REGION Network 23: AXIS W21 MOVE AXIS AND FEED HOLD CONDITIONS
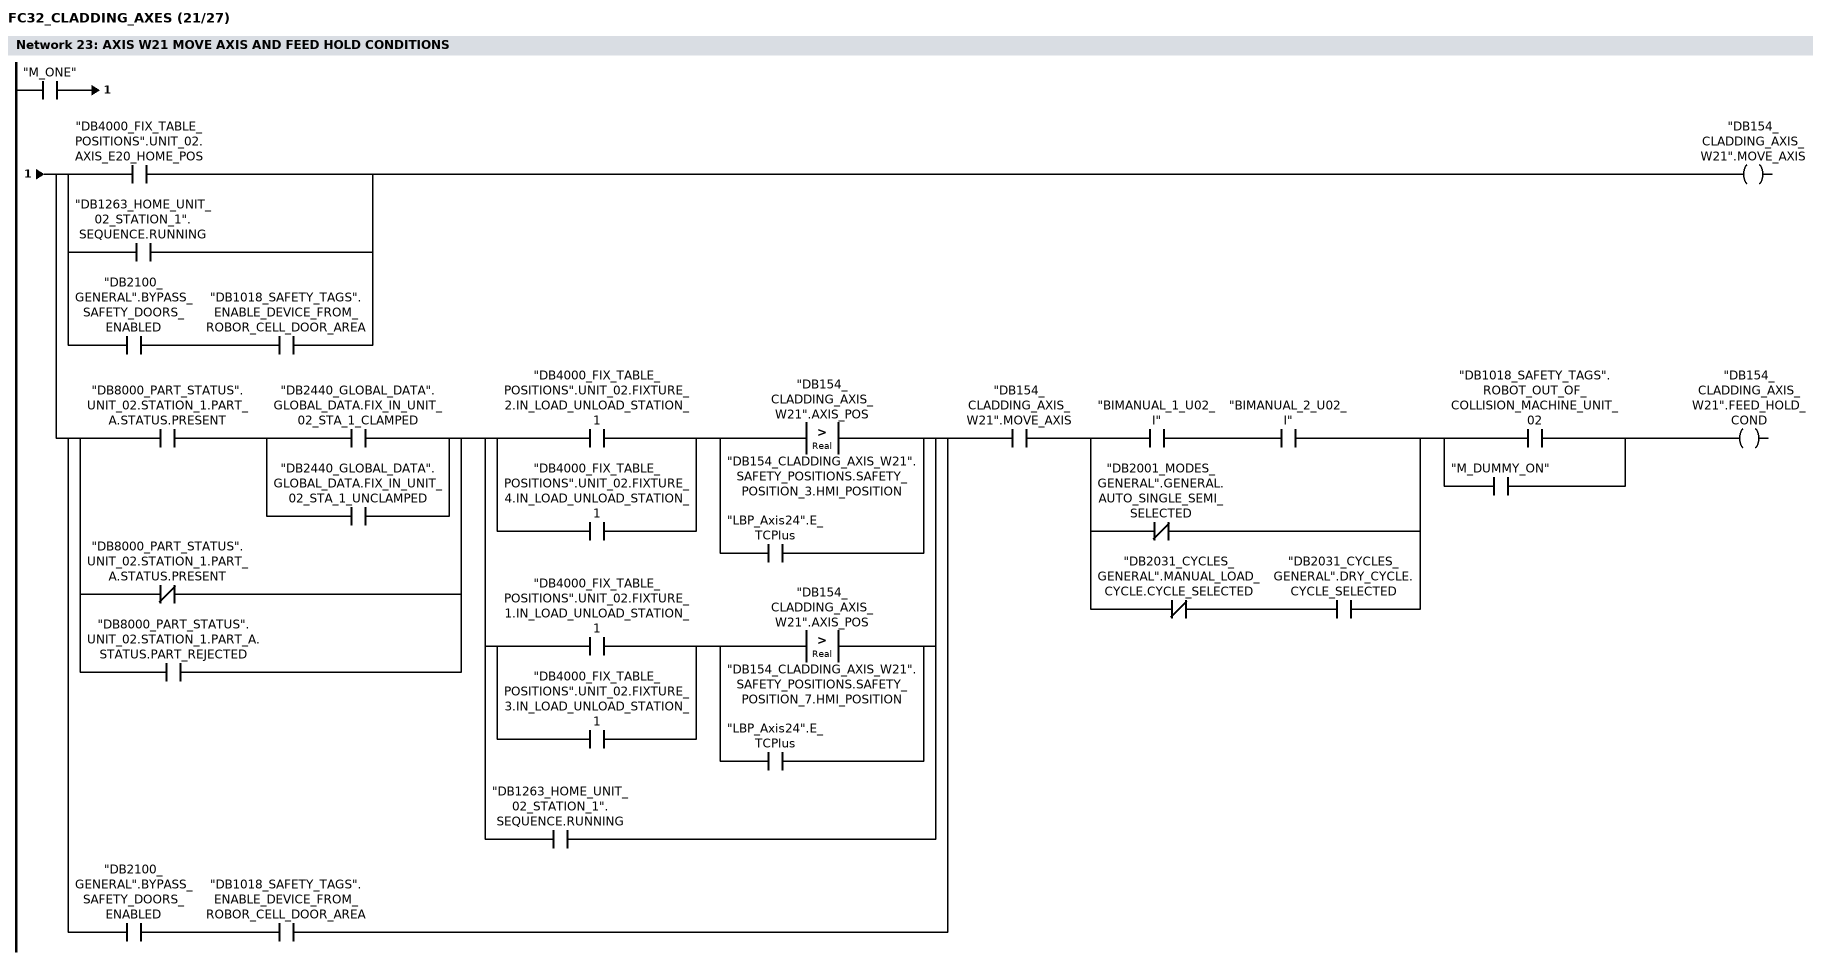
   RUNG wire#powerrail
      Contact( "M_ONE" )
      wire#w1
      Contact( "DB4000_FIX_TABLE_POSITIONS".UNIT_02.AXIS_E20_HOME_POS )
      wire#w2
      Coil( "DB154_CLADDING_AXIS_W21".MOVE_AXIS )
   END_RUNG
   RUNG wire#w1
      Contact( "DB1263_HOME_UNIT_02_STATION_1".SEQUENCE.RUNNING )
   END_RUNG wire#w2
   RUNG wire#w1
      Contact( "DB2100_GENERAL".BYPASS_SAFETY_DOORS_ENABLED )
      Contact( "DB1018_SAFETY_TAGS".ENABLE_DEVICE_FROM_ROBOR_CELL_DOOR_AREA )
   END_RUNG wire#w2
   RUNG wire#w1
      Contact( "DB8000_PART_STATUS".UNIT_02.STATION_1.PART_A.STATUS.PRESENT )
      wire#w3
      Contact( "DB2440_GLOBAL_DATA".GLOBAL_DATA.FIX_IN_UNIT_02_STA_1_CLAMPED )
      wire#w4
      Contact( "DB4000_FIX_TABLE_POSITIONS".UNIT_02.FIXTURE_2.IN_LOAD_UNLOAD_STATION_1 )
      wire#w5
      { S7_Templates := "SrcType := Real" } GT_Contact(in1 := "DB154_CLADDING_AXIS_W21".AXIS_POS, in2 := "DB154_CLADDING_AXIS_W21".SAFETY_POSITIONS.SAFETY_POSITION_3.HMI_POSITION)
      wire#w6
      Contact( "DB154_CLADDING_AXIS_W21".MOVE_AXIS )
      wire#w8
      Contact( "BIMANUAL_1_U02_I" )
      Contact( "BIMANUAL_2_U02_I" )
      wire#w9
      Contact( "DB1018_SAFETY_TAGS".ROBOT_OUT_OF_COLLISION_MACHINE_UNIT_02 )
      wire#w10
      Coil( "DB154_CLADDING_AXIS_W21".FEED_HOLD_COND )
   END_RUNG
   RUNG wire#w3
      Contact( "DB2440_GLOBAL_DATA".GLOBAL_DATA.FIX_IN_UNIT_02_STA_1_UNCLAMPED )
   END_RUNG wire#w4
   RUNG wire#w1
      I_Contact( "DB8000_PART_STATUS".UNIT_02.STATION_1.PART_A.STATUS.PRESENT )
   END_RUNG wire#w4
   RUNG wire#w1
      Contact( "DB8000_PART_STATUS".UNIT_02.STATION_1.PART_A.STATUS.PART_REJECTED )
   END_RUNG wire#w4
   RUNG wire#w4
      Contact( "DB4000_FIX_TABLE_POSITIONS".UNIT_02.FIXTURE_4.IN_LOAD_UNLOAD_STATION_1 )
   END_RUNG wire#w5
   RUNG wire#w5
      Contact( "LBP_Axis24".E_TCPlus )
   END_RUNG wire#w6
   RUNG wire#w4
      Contact( "DB4000_FIX_TABLE_POSITIONS".UNIT_02.FIXTURE_1.IN_LOAD_UNLOAD_STATION_1 )
      wire#w7
      { S7_Templates := "SrcType := Real" } GT_Contact(in1 := "DB154_CLADDING_AXIS_W21".AXIS_POS, in2 := "DB154_CLADDING_AXIS_W21".SAFETY_POSITIONS.SAFETY_POSITION_7.HMI_POSITION)
   END_RUNG wire#w6
   RUNG wire#w4
      Contact( "DB4000_FIX_TABLE_POSITIONS".UNIT_02.FIXTURE_3.IN_LOAD_UNLOAD_STATION_1 )
   END_RUNG wire#w7
   RUNG wire#w7
      Contact( "LBP_Axis24".E_TCPlus )
   END_RUNG wire#w6
   RUNG wire#w4
      Contact( "DB1263_HOME_UNIT_02_STATION_1".SEQUENCE.RUNNING )
   END_RUNG wire#w6
   RUNG wire#w1
      Contact( "DB2100_GENERAL".BYPASS_SAFETY_DOORS_ENABLED )
      Contact( "DB1018_SAFETY_TAGS".ENABLE_DEVICE_FROM_ROBOR_CELL_DOOR_AREA )
   END_RUNG wire#w6
   RUNG wire#w8
      I_Contact( "DB2001_MODES_GENERAL".GENERAL.AUTO_SINGLE_SEMI_SELECTED )
   END_RUNG wire#w9
   RUNG wire#w8
      I_Contact( "DB2031_CYCLES_GENERAL".MANUAL_LOAD_CYCLE.CYCLE_SELECTED )
      Contact( "DB2031_CYCLES_GENERAL".DRY_CYCLE.CYCLE_SELECTED )
   END_RUNG wire#w9
   RUNG wire#w9
      Contact( "M_DUMMY_ON" )
   END_RUNG wire#w10
   // the same network as SCL:
   "DB154_CLADDING_AXIS_W21".MOVE_AXIS := "M_ONE" AND ("DB4000_FIX_TABLE_POSITIONS".UNIT_02.AXIS_E20_HOME_POS OR "DB1263_HOME_UNIT_02_STATION_1".SEQUENCE.RUNNING OR ("DB2100_GENERAL".BYPASS_SAFETY_DOORS_ENABLED AND "DB1018_SAFETY_TAGS".ENABLE_DEVICE_FROM_ROBOR_CELL_DOOR_AREA));
   "DB154_CLADDING_AXIS_W21".FEED_HOLD_COND := "M_ONE" AND (((("DB8000_PART_STATUS".UNIT_02.STATION_1.PART_A.STATUS.PRESENT AND ("DB2440_GLOBAL_DATA".GLOBAL_DATA.FIX_IN_UNIT_02_STA_1_CLAMPED OR "DB2440_GLOBAL_DATA".GLOBAL_DATA.FIX_IN_UNIT_02_STA_1_UNCLAMPED)) OR NOT "DB8000_PART_STATUS".UNIT_02.STATION_1.PART_A.STATUS.PRESENT OR "DB8000_PART_STATUS".UNIT_02.STATION_1.PART_A.STATUS.PART_REJECTED) AND ((("DB4000_FIX_TABLE_POSITIONS".UNIT_02.FIXTURE_2.IN_LOAD_UNLOAD_STATION_1 OR "DB4000_FIX_TABLE_POSITIONS".UNIT_02.FIXTURE_4.IN_LOAD_UNLOAD_STATION_1) AND (("DB154_CLADDING_AXIS_W21".AXIS_POS > "DB154_CLADDING_AXIS_W21".SAFETY_POSITIONS.SAFETY_POSITION_3.HMI_POSITION) OR "LBP_Axis24".E_TCPlus)) OR (("DB4000_FIX_TABLE_POSITIONS".UNIT_02.FIXTURE_1.IN_LOAD_UNLOAD_STATION_1 OR "DB4000_FIX_TABLE_POSITIONS".UNIT_02.FIXTURE_3.IN_LOAD_UNLOAD_STATION_1) AND (("DB154_CLADDING_AXIS_W21".AXIS_POS > "DB154_CLADDING_AXIS_W21".SAFETY_POSITIONS.SAFETY_POSITION_7.HMI_POSITION) OR "LBP_Axis24".E_TCPlus)) OR "DB1263_HOME_UNIT_02_STATION_1".SEQUENCE.RUNNING)) OR ("DB2100_GENERAL".BYPASS_SAFETY_DOORS_ENABLED AND "DB1018_SAFETY_TAGS".ENABLE_DEVICE_FROM_ROBOR_CELL_DOOR_AREA)) AND "DB154_CLADDING_AXIS_W21".MOVE_AXIS AND (("BIMANUAL_1_U02_I" AND "BIMANUAL_2_U02_I") OR NOT "DB2001_MODES_GENERAL".GENERAL.AUTO_SINGLE_SEMI_SELECTED OR (NOT "DB2031_CYCLES_GENERAL".MANUAL_LOAD_CYCLE.CYCLE_SELECTED AND "DB2031_CYCLES_GENERAL".DRY_CYCLE.CYCLE_SELECTED)) AND ("DB1018_SAFETY_TAGS".ROBOT_OUT_OF_COLLISION_MACHINE_UNIT_02 OR "M_DUMMY_ON");
END_REGION

REGION Network 24: CALL FB32 AXIS W21
   // 2#0000_0001 OPTIONS 0 BIT 0 MEASURING SYSTEM 2 OPTION
   // 2#0000_0010 OPTIONS 0 BIT 1 ENABLE FC18 OPTION
   // 2#0000_0100 OPTIONS 0 BIT 2 FC18 EXTERNAL POSITION OPTION
   // 2#0000_1000 OPTIONS 0 BIT 3 AXIS B ENABLE FAULTS OPTION
   // 2#0001_0000 OPTIONS 0 BIT 4 SPARE OPTION
   // 2#0010_0000 OPTIONS 0 BIT 5 SPARE OPTION
   // 2#0100_0000 OPTIONS 0 BIT 6 SPARE OPTION
   // 2#1000_0000 OPTIONS 0 BIT 7 SPARE OPTION
   // 
   // 2#0000_0001 OPTIONS 1 BIT 0 AXIS ROLLER OPTION
   // 2#0000_0010 OPTIONS 1 BIT 1 MASTER AXIS OPTION
   // 2#0000_0100 OPTIONS 1 BIT 2 SLAVE AXIS OPTION
   // 2#0000_1000 OPTIONS 1 BIT 3 MASTER-SLAVE AXES INDEPENDENT MOVEMENT WITH HT10 OPTION
   // 2#0001_0000 OPTIONS 1 BIT 4 GANTRY MODE MASTER AXIS OPTION
   // 2#0010_0000 OPTIONS 1 BIT 5 SPARE OPTION
   // 2#0100_0000 OPTIONS 1 BIT 6 SPARE OPTION
   // 2#1000_0000 OPTIONS 1 BIT 7 SPARE OPTION
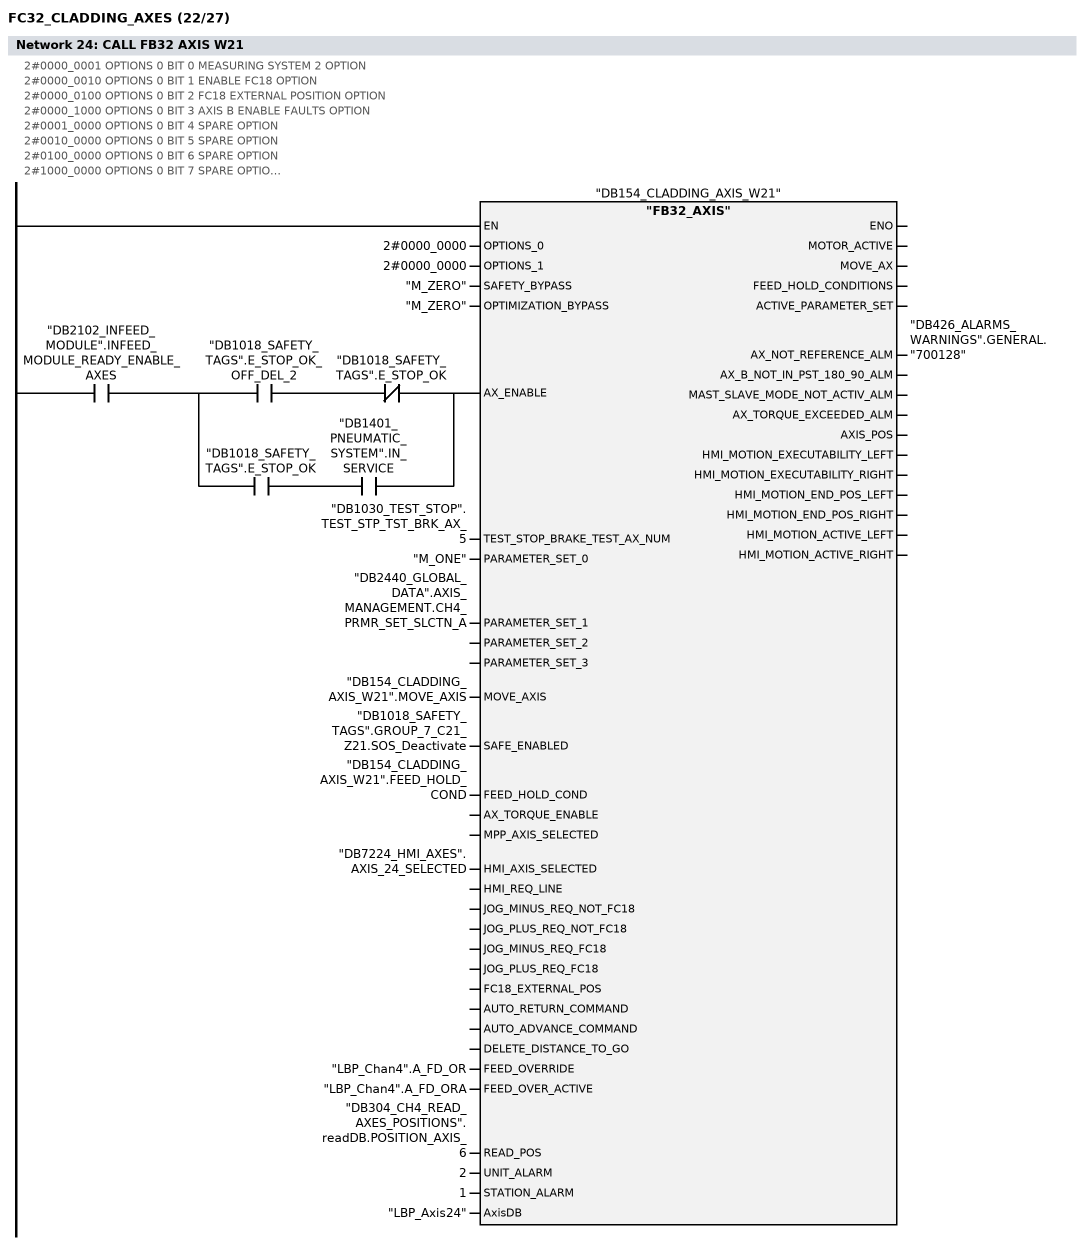
   RUNG wire#powerrail
      "DB154_CLADDING_AXIS_W21"(AX_ENABLE := wire#w2, OPTIONS_0 := 2#0000_0000, OPTIONS_1 := 2#0000_0000, SAFETY_BYPASS := "M_ZERO", OPTIMIZATION_BYPASS := "M_ZERO", TEST_STOP_BRAKE_TEST_AX_NUM := "DB1030_TEST_STOP".TEST_STP_TST_BRK_AX_5, PARAMETER_SET_0 := "M_ONE", PARAMETER_SET_1 := "DB2440_GLOBAL_DATA".AXIS_MANAGEMENT.CH4_PRMR_SET_SLCTN_A, PARAMETER_SET_2 :=, PARAMETER_SET_3 :=, MOVE_AXIS := "DB154_CLADDING_AXIS_W21".MOVE_AXIS, SAFE_ENABLED := "DB1018_SAFETY_TAGS".GROUP_7_C21_Z21.SOS_Deactivate, FEED_HOLD_COND := "DB154_CLADDING_AXIS_W21".FEED_HOLD_COND, AX_TORQUE_ENABLE :=, MPP_AXIS_SELECTED :=, HMI_AXIS_SELECTED := "DB7224_HMI_AXES".AXIS_24_SELECTED, HMI_REQ_LINE :=, JOG_MINUS_REQ_NOT_FC18 :=, JOG_PLUS_REQ_NOT_FC18 :=, JOG_MINUS_REQ_FC18 :=, JOG_PLUS_REQ_FC18 :=, FC18_EXTERNAL_POS :=, AUTO_RETURN_COMMAND :=, AUTO_ADVANCE_COMMAND :=, DELETE_DISTANCE_TO_GO :=, FEED_OVERRIDE := "LBP_Chan4".A_FD_OR, FEED_OVER_ACTIVE := "LBP_Chan4".A_FD_ORA, READ_POS := "DB304_CH4_READ_AXES_POSITIONS".readDB.POSITION_AXIS_6, UNIT_ALARM := 2, STATION_ALARM := 1, AxisDB := "LBP_Axis24", MOTOR_ACTIVE =>, MOVE_AX =>, FEED_HOLD_CONDITIONS =>, ACTIVE_PARAMETER_SET =>, AX_NOT_REFERENCE_ALM => "DB426_ALARMS_WARNINGS".GENERAL."700128", AX_B_NOT_IN_PST_180_90_ALM =>, MAST_SLAVE_MODE_NOT_ACTIV_ALM =>, AX_TORQUE_EXCEEDED_ALM =>, AXIS_POS =>, HMI_MOTION_EXECUTABILITY_LEFT =>, HMI_MOTION_EXECUTABILITY_RIGHT =>, HMI_MOTION_END_POS_LEFT =>, HMI_MOTION_END_POS_RIGHT =>, HMI_MOTION_ACTIVE_LEFT =>, HMI_MOTION_ACTIVE_RIGHT =>)
   END_RUNG
   RUNG wire#powerrail
      Contact( "DB2102_INFEED_MODULE".INFEED_MODULE_READY_ENABLE_AXES )
      wire#w1
      Contact( "DB1018_SAFETY_TAGS".E_STOP_OK_OFF_DEL_2 )
      I_Contact( "DB1018_SAFETY_TAGS".E_STOP_OK )
   END_RUNG wire#w2
   RUNG wire#w1
      Contact( "DB1018_SAFETY_TAGS".E_STOP_OK )
      Contact( "DB1401_PNEUMATIC_SYSTEM".IN_SERVICE )
   END_RUNG wire#w2
   // the same network as SCL:
   "DB154_CLADDING_AXIS_W21"(OPTIONS_0 := 2#0000_0000,   // "FB32_AXIS"
                           OPTIONS_1 := 2#0000_0000,
                           SAFETY_BYPASS := "M_ZERO",
                           OPTIMIZATION_BYPASS := "M_ZERO",
                           AX_ENABLE := "DB2102_INFEED_MODULE".INFEED_MODULE_READY_ENABLE_AXES AND (("DB1018_SAFETY_TAGS".E_STOP_OK_OFF_DEL_2 AND NOT "DB1018_SAFETY_TAGS".E_STOP_OK) OR ("DB1018_SAFETY_TAGS".E_STOP_OK AND "DB1401_PNEUMATIC_SYSTEM".IN_SERVICE)),
                           TEST_STOP_BRAKE_TEST_AX_NUM := "DB1030_TEST_STOP".TEST_STP_TST_BRK_AX_5,
                           PARAMETER_SET_0 := "M_ONE",
                           PARAMETER_SET_1 := "DB2440_GLOBAL_DATA".AXIS_MANAGEMENT.CH4_PRMR_SET_SLCTN_A,
                           MOVE_AXIS := "DB154_CLADDING_AXIS_W21".MOVE_AXIS,
                           SAFE_ENABLED := "DB1018_SAFETY_TAGS".GROUP_7_C21_Z21.SOS_Deactivate,
                           FEED_HOLD_COND := "DB154_CLADDING_AXIS_W21".FEED_HOLD_COND,
                           HMI_AXIS_SELECTED := "DB7224_HMI_AXES".AXIS_24_SELECTED,
                           FEED_OVERRIDE := "LBP_Chan4".A_FD_OR,
                           FEED_OVER_ACTIVE := "LBP_Chan4".A_FD_ORA,
                           READ_POS := "DB304_CH4_READ_AXES_POSITIONS".readDB.POSITION_AXIS_6,
                           UNIT_ALARM := 2,
                           STATION_ALARM := 1,
                           AxisDB := "LBP_Axis24",
                           AX_NOT_REFERENCE_ALM => "DB426_ALARMS_WARNINGS".GENERAL."700128");
END_REGION

REGION Network 25: AXIS W21 OPERATOR HELP
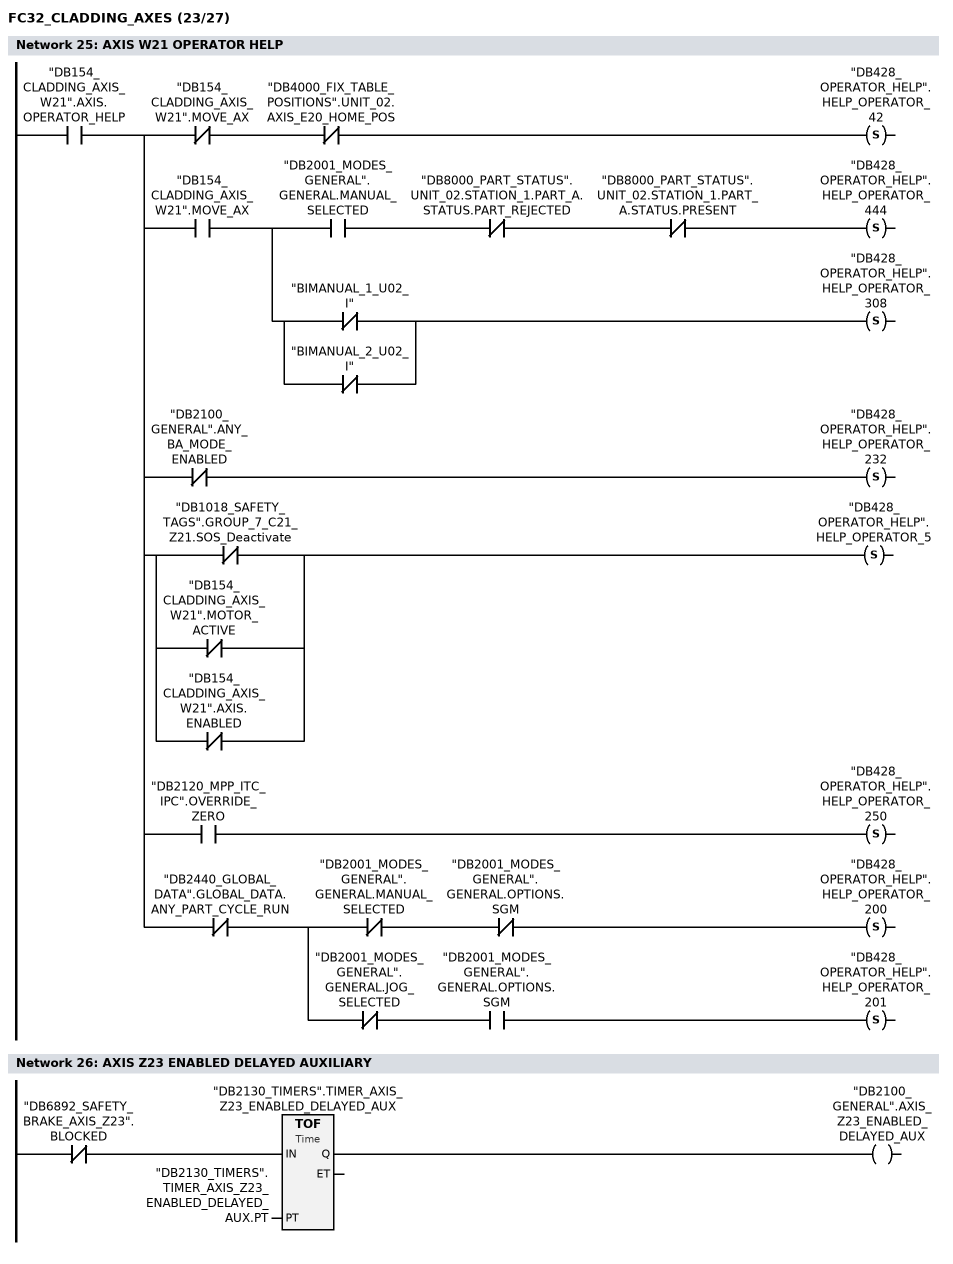
   RUNG wire#powerrail
      Contact( "DB154_CLADDING_AXIS_W21".AXIS.OPERATOR_HELP )
      wire#w1
      I_Contact( "DB154_CLADDING_AXIS_W21".MOVE_AX )
      I_Contact( "DB4000_FIX_TABLE_POSITIONS".UNIT_02.AXIS_E20_HOME_POS )
      S_Coil( "DB428_OPERATOR_HELP".HELP_OPERATOR_42 )
   END_RUNG
   RUNG wire#w1
      Contact( "DB154_CLADDING_AXIS_W21".MOVE_AX )
      wire#w2
      Contact( "DB2001_MODES_GENERAL".GENERAL.MANUAL_SELECTED )
      I_Contact( "DB8000_PART_STATUS".UNIT_02.STATION_1.PART_A.STATUS.PART_REJECTED )
      I_Contact( "DB8000_PART_STATUS".UNIT_02.STATION_1.PART_A.STATUS.PRESENT )
      S_Coil( "DB428_OPERATOR_HELP".HELP_OPERATOR_444 )
   END_RUNG
   RUNG wire#w2
      I_Contact( "BIMANUAL_1_U02_I" )
      wire#w3
      S_Coil( "DB428_OPERATOR_HELP".HELP_OPERATOR_308 )
   END_RUNG
   RUNG wire#w2
      I_Contact( "BIMANUAL_2_U02_I" )
   END_RUNG wire#w3
   RUNG wire#w1
      I_Contact( "DB2100_GENERAL".ANY_BA_MODE_ENABLED )
      S_Coil( "DB428_OPERATOR_HELP".HELP_OPERATOR_232 )
   END_RUNG
   RUNG wire#w1
      I_Contact( "DB1018_SAFETY_TAGS".GROUP_7_C21_Z21.SOS_Deactivate )
      wire#w4
      S_Coil( "DB428_OPERATOR_HELP".HELP_OPERATOR_5 )
   END_RUNG
   RUNG wire#w1
      I_Contact( "DB154_CLADDING_AXIS_W21".MOTOR_ACTIVE )
   END_RUNG wire#w4
   RUNG wire#w1
      I_Contact( "DB154_CLADDING_AXIS_W21".AXIS.ENABLED )
   END_RUNG wire#w4
   RUNG wire#w1
      Contact( "DB2120_MPP_ITC_IPC".OVERRIDE_ZERO )
      S_Coil( "DB428_OPERATOR_HELP".HELP_OPERATOR_250 )
   END_RUNG
   RUNG wire#w1
      I_Contact( "DB2440_GLOBAL_DATA".GLOBAL_DATA.ANY_PART_CYCLE_RUN )
      wire#w5
      I_Contact( "DB2001_MODES_GENERAL".GENERAL.MANUAL_SELECTED )
      I_Contact( "DB2001_MODES_GENERAL".GENERAL.OPTIONS.SGM )
      S_Coil( "DB428_OPERATOR_HELP".HELP_OPERATOR_200 )
   END_RUNG
   RUNG wire#w5
      I_Contact( "DB2001_MODES_GENERAL".GENERAL.JOG_SELECTED )
      Contact( "DB2001_MODES_GENERAL".GENERAL.OPTIONS.SGM )
      S_Coil( "DB428_OPERATOR_HELP".HELP_OPERATOR_201 )
   END_RUNG
   // the same network as SCL:
   IF "DB154_CLADDING_AXIS_W21".AXIS.OPERATOR_HELP AND NOT "DB154_CLADDING_AXIS_W21".MOVE_AX AND NOT "DB4000_FIX_TABLE_POSITIONS".UNIT_02.AXIS_E20_HOME_POS THEN
       "DB428_OPERATOR_HELP".HELP_OPERATOR_42 := TRUE;
   END_IF;
   #_w1 := "DB154_CLADDING_AXIS_W21".AXIS.OPERATOR_HELP AND "DB154_CLADDING_AXIS_W21".MOVE_AX;
   IF #_w1 AND "DB2001_MODES_GENERAL".GENERAL.MANUAL_SELECTED AND NOT "DB8000_PART_STATUS".UNIT_02.STATION_1.PART_A.STATUS.PART_REJECTED AND NOT "DB8000_PART_STATUS".UNIT_02.STATION_1.PART_A.STATUS.PRESENT THEN
       "DB428_OPERATOR_HELP".HELP_OPERATOR_444 := TRUE;
   END_IF;
   IF #_w1 AND (NOT "BIMANUAL_1_U02_I" OR NOT "BIMANUAL_2_U02_I") THEN
       "DB428_OPERATOR_HELP".HELP_OPERATOR_308 := TRUE;
   END_IF;
   IF "DB154_CLADDING_AXIS_W21".AXIS.OPERATOR_HELP AND NOT "DB2100_GENERAL".ANY_BA_MODE_ENABLED THEN
       "DB428_OPERATOR_HELP".HELP_OPERATOR_232 := TRUE;
   END_IF;
   IF "DB154_CLADDING_AXIS_W21".AXIS.OPERATOR_HELP AND (NOT "DB1018_SAFETY_TAGS".GROUP_7_C21_Z21.SOS_Deactivate OR NOT "DB154_CLADDING_AXIS_W21".MOTOR_ACTIVE OR NOT "DB154_CLADDING_AXIS_W21".AXIS.ENABLED) THEN
       "DB428_OPERATOR_HELP".HELP_OPERATOR_5 := TRUE;
   END_IF;
   IF "DB154_CLADDING_AXIS_W21".AXIS.OPERATOR_HELP AND "DB2120_MPP_ITC_IPC".OVERRIDE_ZERO THEN
       "DB428_OPERATOR_HELP".HELP_OPERATOR_250 := TRUE;
   END_IF;
   #_w2 := "DB154_CLADDING_AXIS_W21".AXIS.OPERATOR_HELP AND NOT "DB2440_GLOBAL_DATA".GLOBAL_DATA.ANY_PART_CYCLE_RUN;
   IF #_w2 AND NOT "DB2001_MODES_GENERAL".GENERAL.MANUAL_SELECTED AND NOT "DB2001_MODES_GENERAL".GENERAL.OPTIONS.SGM THEN
       "DB428_OPERATOR_HELP".HELP_OPERATOR_200 := TRUE;
   END_IF;
   IF #_w2 AND NOT "DB2001_MODES_GENERAL".GENERAL.JOG_SELECTED AND "DB2001_MODES_GENERAL".GENERAL.OPTIONS.SGM THEN
       "DB428_OPERATOR_HELP".HELP_OPERATOR_201 := TRUE;
   END_IF;
END_REGION

REGION Network 26: AXIS Z23 ENABLED DELAYED AUXILIARY
   RUNG wire#powerrail
      I_Contact( "DB6892_SAFETY_BRAKE_AXIS_Z23".BLOCKED )
      { S7_Templates := "time_type := Time" } "DB2130_TIMERS".TIMER_AXIS_Z23_ENABLED_DELAYED_AUX.TOF(pt := "DB2130_TIMERS".TIMER_AXIS_Z23_ENABLED_DELAYED_AUX.PT, et =>)
      Coil( "DB2100_GENERAL".AXIS_Z23_ENABLED_DELAYED_AUX )
   END_RUNG
   // the same network as SCL:
   "DB2130_TIMERS".TIMER_AXIS_Z23_ENABLED_DELAYED_AUX.TOF(IN := NOT "DB6892_SAFETY_BRAKE_AXIS_Z23".BLOCKED,
                           PT := "DB2130_TIMERS".TIMER_AXIS_Z23_ENABLED_DELAYED_AUX.PT);
   "DB2100_GENERAL".AXIS_Z23_ENABLED_DELAYED_AUX := "DB2130_TIMERS".TIMER_AXIS_Z23_ENABLED_DELAYED_AUX.Q;
END_REGION

REGION Network 27: AXIS Z23 MOVE AXIS AND FEED HOLD CONDITIONS
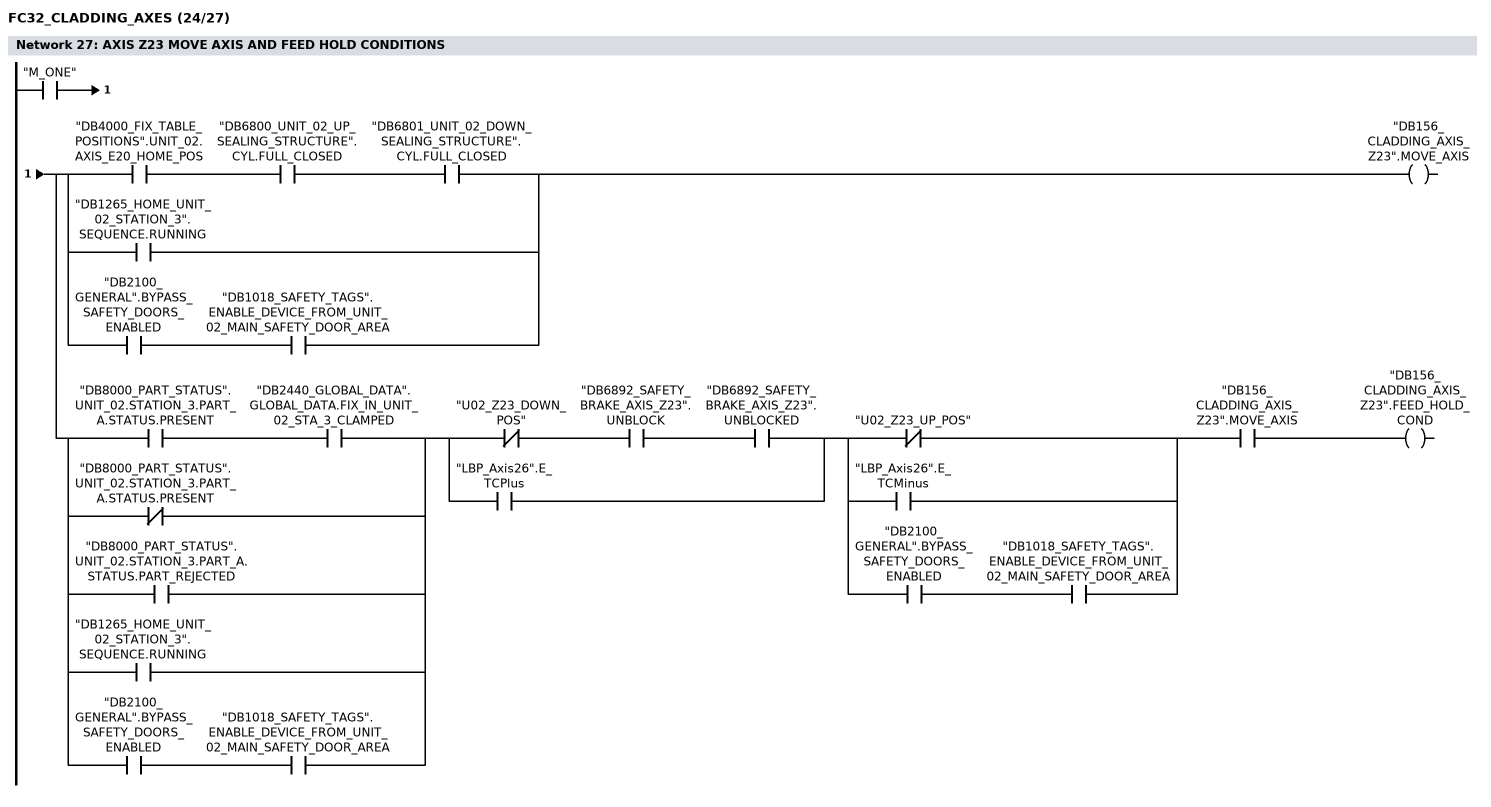
   RUNG wire#powerrail
      Contact( "M_ONE" )
      wire#w1
      Contact( "DB4000_FIX_TABLE_POSITIONS".UNIT_02.AXIS_E20_HOME_POS )
      Contact( "DB6800_UNIT_02_UP_SEALING_STRUCTURE".CYL.FULL_CLOSED )
      Contact( "DB6801_UNIT_02_DOWN_SEALING_STRUCTURE".CYL.FULL_CLOSED )
      wire#w2
      Coil( "DB156_CLADDING_AXIS_Z23".MOVE_AXIS )
   END_RUNG
   RUNG wire#w1
      Contact( "DB1265_HOME_UNIT_02_STATION_3".SEQUENCE.RUNNING )
   END_RUNG wire#w2
   RUNG wire#w1
      Contact( "DB2100_GENERAL".BYPASS_SAFETY_DOORS_ENABLED )
      Contact( "DB1018_SAFETY_TAGS".ENABLE_DEVICE_FROM_UNIT_02_MAIN_SAFETY_DOOR_AREA )
   END_RUNG wire#w2
   RUNG wire#w1
      Contact( "DB8000_PART_STATUS".UNIT_02.STATION_3.PART_A.STATUS.PRESENT )
      Contact( "DB2440_GLOBAL_DATA".GLOBAL_DATA.FIX_IN_UNIT_02_STA_3_CLAMPED )
      wire#w3
      I_Contact( "U02_Z23_DOWN_POS" )
      Contact( "DB6892_SAFETY_BRAKE_AXIS_Z23".UNBLOCK )
      Contact( "DB6892_SAFETY_BRAKE_AXIS_Z23".UNBLOCKED )
      wire#w4
      I_Contact( "U02_Z23_UP_POS" )
      wire#w5
      Contact( "DB156_CLADDING_AXIS_Z23".MOVE_AXIS )
      Coil( "DB156_CLADDING_AXIS_Z23".FEED_HOLD_COND )
   END_RUNG
   RUNG wire#w1
      I_Contact( "DB8000_PART_STATUS".UNIT_02.STATION_3.PART_A.STATUS.PRESENT )
   END_RUNG wire#w3
   RUNG wire#w1
      Contact( "DB8000_PART_STATUS".UNIT_02.STATION_3.PART_A.STATUS.PART_REJECTED )
   END_RUNG wire#w3
   RUNG wire#w1
      Contact( "DB1265_HOME_UNIT_02_STATION_3".SEQUENCE.RUNNING )
   END_RUNG wire#w3
   RUNG wire#w1
      Contact( "DB2100_GENERAL".BYPASS_SAFETY_DOORS_ENABLED )
      Contact( "DB1018_SAFETY_TAGS".ENABLE_DEVICE_FROM_UNIT_02_MAIN_SAFETY_DOOR_AREA )
   END_RUNG wire#w3
   RUNG wire#w3
      Contact( "LBP_Axis26".E_TCPlus )
   END_RUNG wire#w4
   RUNG wire#w4
      Contact( "LBP_Axis26".E_TCMinus )
   END_RUNG wire#w5
   RUNG wire#w4
      Contact( "DB2100_GENERAL".BYPASS_SAFETY_DOORS_ENABLED )
      Contact( "DB1018_SAFETY_TAGS".ENABLE_DEVICE_FROM_UNIT_02_MAIN_SAFETY_DOOR_AREA )
   END_RUNG wire#w5
   // the same network as SCL:
   "DB156_CLADDING_AXIS_Z23".MOVE_AXIS := "M_ONE" AND (("DB4000_FIX_TABLE_POSITIONS".UNIT_02.AXIS_E20_HOME_POS AND "DB6800_UNIT_02_UP_SEALING_STRUCTURE".CYL.FULL_CLOSED AND "DB6801_UNIT_02_DOWN_SEALING_STRUCTURE".CYL.FULL_CLOSED) OR "DB1265_HOME_UNIT_02_STATION_3".SEQUENCE.RUNNING OR ("DB2100_GENERAL".BYPASS_SAFETY_DOORS_ENABLED AND "DB1018_SAFETY_TAGS".ENABLE_DEVICE_FROM_UNIT_02_MAIN_SAFETY_DOOR_AREA));
   "DB156_CLADDING_AXIS_Z23".FEED_HOLD_COND := "M_ONE" AND (("DB8000_PART_STATUS".UNIT_02.STATION_3.PART_A.STATUS.PRESENT AND "DB2440_GLOBAL_DATA".GLOBAL_DATA.FIX_IN_UNIT_02_STA_3_CLAMPED) OR NOT "DB8000_PART_STATUS".UNIT_02.STATION_3.PART_A.STATUS.PRESENT OR "DB8000_PART_STATUS".UNIT_02.STATION_3.PART_A.STATUS.PART_REJECTED OR "DB1265_HOME_UNIT_02_STATION_3".SEQUENCE.RUNNING OR ("DB2100_GENERAL".BYPASS_SAFETY_DOORS_ENABLED AND "DB1018_SAFETY_TAGS".ENABLE_DEVICE_FROM_UNIT_02_MAIN_SAFETY_DOOR_AREA)) AND ((NOT "U02_Z23_DOWN_POS" AND "DB6892_SAFETY_BRAKE_AXIS_Z23".UNBLOCK AND "DB6892_SAFETY_BRAKE_AXIS_Z23".UNBLOCKED) OR "LBP_Axis26".E_TCPlus) AND (NOT "U02_Z23_UP_POS" OR "LBP_Axis26".E_TCMinus OR ("DB2100_GENERAL".BYPASS_SAFETY_DOORS_ENABLED AND "DB1018_SAFETY_TAGS".ENABLE_DEVICE_FROM_UNIT_02_MAIN_SAFETY_DOOR_AREA)) AND "DB156_CLADDING_AXIS_Z23".MOVE_AXIS;
END_REGION

REGION Network 28: CALL FB32 AXIS Z23
   // 2#0000_0001 OPTIONS 0 BIT 0 MEASURING SYSTEM 2 OPTION
   // 2#0000_0010 OPTIONS 0 BIT 1 ENABLE FC18 OPTION
   // 2#0000_0100 OPTIONS 0 BIT 2 FC18 EXTERNAL POSITION OPTION
   // 2#0000_1000 OPTIONS 0 BIT 3 AXIS B ENABLE FAULTS OPTION
   // 2#0001_0000 OPTIONS 0 BIT 4 SPARE OPTION
   // 2#0010_0000 OPTIONS 0 BIT 5 SPARE OPTION
   // 2#0100_0000 OPTIONS 0 BIT 6 SPARE OPTION
   // 2#1000_0000 OPTIONS 0 BIT 7 SPARE OPTION
   // 
   // 2#0000_0001 OPTIONS 1 BIT 0 AXIS ROLLER OPTION
   // 2#0000_0010 OPTIONS 1 BIT 1 MASTER AXIS OPTION
   // 2#0000_0100 OPTIONS 1 BIT 2 SLAVE AXIS OPTION
   // 2#0000_1000 OPTIONS 1 BIT 3 MASTER-SLAVE AXES INDEPENDENT MOVEMENT WITH HT10 OPTION
   // 2#0001_0000 OPTIONS 1 BIT 4 GANTRY MODE MASTER AXIS OPTION
   // 2#0010_0000 OPTIONS 1 BIT 5 SPARE OPTION
   // 2#0100_0000 OPTIONS 1 BIT 6 SPARE OPTION
   // 2#1000_0000 OPTIONS 1 BIT 7 SPARE OPTION
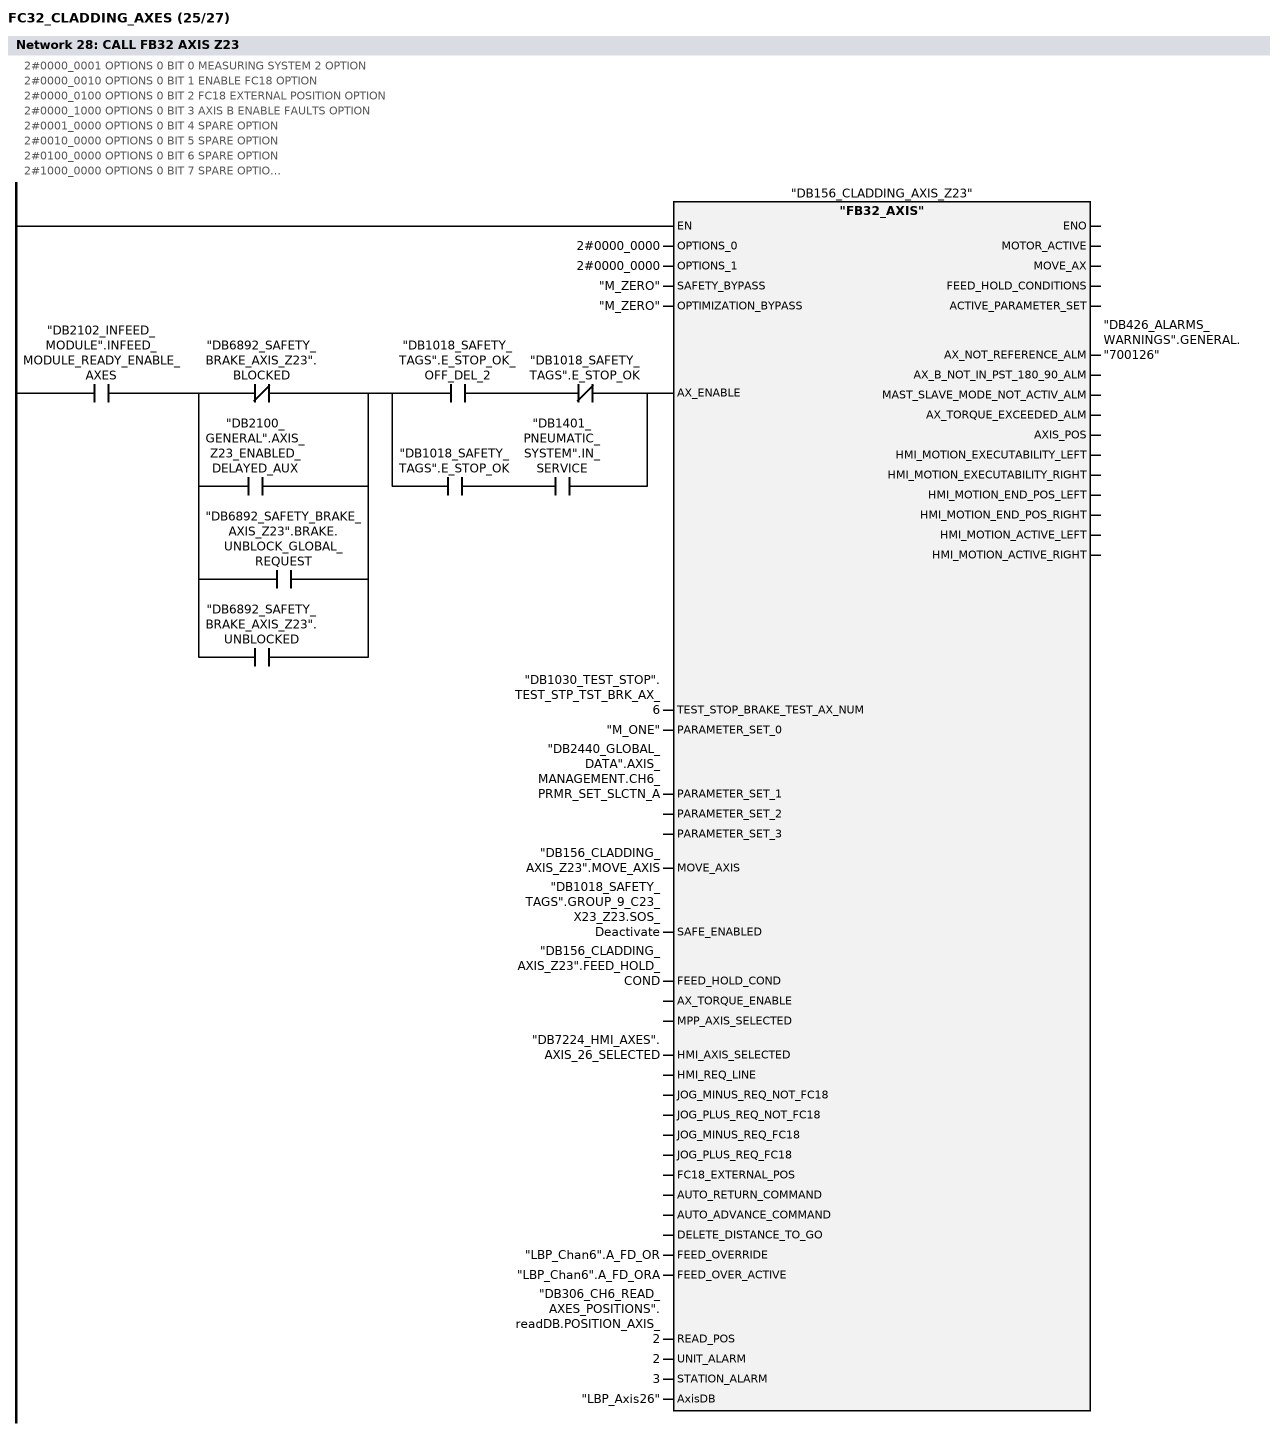
   RUNG wire#powerrail
      "DB156_CLADDING_AXIS_Z23"(AX_ENABLE := wire#w3, OPTIONS_0 := 2#0000_0000, OPTIONS_1 := 2#0000_0000, SAFETY_BYPASS := "M_ZERO", OPTIMIZATION_BYPASS := "M_ZERO", TEST_STOP_BRAKE_TEST_AX_NUM := "DB1030_TEST_STOP".TEST_STP_TST_BRK_AX_6, PARAMETER_SET_0 := "M_ONE", PARAMETER_SET_1 := "DB2440_GLOBAL_DATA".AXIS_MANAGEMENT.CH6_PRMR_SET_SLCTN_A, PARAMETER_SET_2 :=, PARAMETER_SET_3 :=, MOVE_AXIS := "DB156_CLADDING_AXIS_Z23".MOVE_AXIS, SAFE_ENABLED := "DB1018_SAFETY_TAGS".GROUP_9_C23_X23_Z23.SOS_Deactivate, FEED_HOLD_COND := "DB156_CLADDING_AXIS_Z23".FEED_HOLD_COND, AX_TORQUE_ENABLE :=, MPP_AXIS_SELECTED :=, HMI_AXIS_SELECTED := "DB7224_HMI_AXES".AXIS_26_SELECTED, HMI_REQ_LINE :=, JOG_MINUS_REQ_NOT_FC18 :=, JOG_PLUS_REQ_NOT_FC18 :=, JOG_MINUS_REQ_FC18 :=, JOG_PLUS_REQ_FC18 :=, FC18_EXTERNAL_POS :=, AUTO_RETURN_COMMAND :=, AUTO_ADVANCE_COMMAND :=, DELETE_DISTANCE_TO_GO :=, FEED_OVERRIDE := "LBP_Chan6".A_FD_OR, FEED_OVER_ACTIVE := "LBP_Chan6".A_FD_ORA, READ_POS := "DB306_CH6_READ_AXES_POSITIONS".readDB.POSITION_AXIS_2, UNIT_ALARM := 2, STATION_ALARM := 3, AxisDB := "LBP_Axis26", MOTOR_ACTIVE =>, MOVE_AX =>, FEED_HOLD_CONDITIONS =>, ACTIVE_PARAMETER_SET =>, AX_NOT_REFERENCE_ALM => "DB426_ALARMS_WARNINGS".GENERAL."700126", AX_B_NOT_IN_PST_180_90_ALM =>, MAST_SLAVE_MODE_NOT_ACTIV_ALM =>, AX_TORQUE_EXCEEDED_ALM =>, AXIS_POS =>, HMI_MOTION_EXECUTABILITY_LEFT =>, HMI_MOTION_EXECUTABILITY_RIGHT =>, HMI_MOTION_END_POS_LEFT =>, HMI_MOTION_END_POS_RIGHT =>, HMI_MOTION_ACTIVE_LEFT =>, HMI_MOTION_ACTIVE_RIGHT =>)
   END_RUNG
   RUNG wire#powerrail
      Contact( "DB2102_INFEED_MODULE".INFEED_MODULE_READY_ENABLE_AXES )
      wire#w1
      I_Contact( "DB6892_SAFETY_BRAKE_AXIS_Z23".BLOCKED )
      wire#w2
      Contact( "DB1018_SAFETY_TAGS".E_STOP_OK_OFF_DEL_2 )
      I_Contact( "DB1018_SAFETY_TAGS".E_STOP_OK )
   END_RUNG wire#w3
   RUNG wire#w1
      Contact( "DB2100_GENERAL".AXIS_Z23_ENABLED_DELAYED_AUX )
   END_RUNG wire#w2
   RUNG wire#w1
      Contact( "DB6892_SAFETY_BRAKE_AXIS_Z23".BRAKE.UNBLOCK_GLOBAL_REQUEST )
   END_RUNG wire#w2
   RUNG wire#w1
      Contact( "DB6892_SAFETY_BRAKE_AXIS_Z23".UNBLOCKED )
   END_RUNG wire#w2
   RUNG wire#w2
      Contact( "DB1018_SAFETY_TAGS".E_STOP_OK )
      Contact( "DB1401_PNEUMATIC_SYSTEM".IN_SERVICE )
   END_RUNG wire#w3
   // the same network as SCL:
   "DB156_CLADDING_AXIS_Z23"(OPTIONS_0 := 2#0000_0000,   // "FB32_AXIS"
                           OPTIONS_1 := 2#0000_0000,
                           SAFETY_BYPASS := "M_ZERO",
                           OPTIMIZATION_BYPASS := "M_ZERO",
                           AX_ENABLE := "DB2102_INFEED_MODULE".INFEED_MODULE_READY_ENABLE_AXES AND (NOT "DB6892_SAFETY_BRAKE_AXIS_Z23".BLOCKED OR "DB2100_GENERAL".AXIS_Z23_ENABLED_DELAYED_AUX OR "DB6892_SAFETY_BRAKE_AXIS_Z23".BRAKE.UNBLOCK_GLOBAL_REQUEST OR "DB6892_SAFETY_BRAKE_AXIS_Z23".UNBLOCKED) AND (("DB1018_SAFETY_TAGS".E_STOP_OK_OFF_DEL_2 AND NOT "DB1018_SAFETY_TAGS".E_STOP_OK) OR ("DB1018_SAFETY_TAGS".E_STOP_OK AND "DB1401_PNEUMATIC_SYSTEM".IN_SERVICE)),
                           TEST_STOP_BRAKE_TEST_AX_NUM := "DB1030_TEST_STOP".TEST_STP_TST_BRK_AX_6,
                           PARAMETER_SET_0 := "M_ONE",
                           PARAMETER_SET_1 := "DB2440_GLOBAL_DATA".AXIS_MANAGEMENT.CH6_PRMR_SET_SLCTN_A,
                           MOVE_AXIS := "DB156_CLADDING_AXIS_Z23".MOVE_AXIS,
                           SAFE_ENABLED := "DB1018_SAFETY_TAGS".GROUP_9_C23_X23_Z23.SOS_Deactivate,
                           FEED_HOLD_COND := "DB156_CLADDING_AXIS_Z23".FEED_HOLD_COND,
                           HMI_AXIS_SELECTED := "DB7224_HMI_AXES".AXIS_26_SELECTED,
                           FEED_OVERRIDE := "LBP_Chan6".A_FD_OR,
                           FEED_OVER_ACTIVE := "LBP_Chan6".A_FD_ORA,
                           READ_POS := "DB306_CH6_READ_AXES_POSITIONS".readDB.POSITION_AXIS_2,
                           UNIT_ALARM := 2,
                           STATION_ALARM := 3,
                           AxisDB := "LBP_Axis26",
                           AX_NOT_REFERENCE_ALM => "DB426_ALARMS_WARNINGS".GENERAL."700126");
END_REGION

REGION Network 29: AXIS Z23 OPERATOR HELP
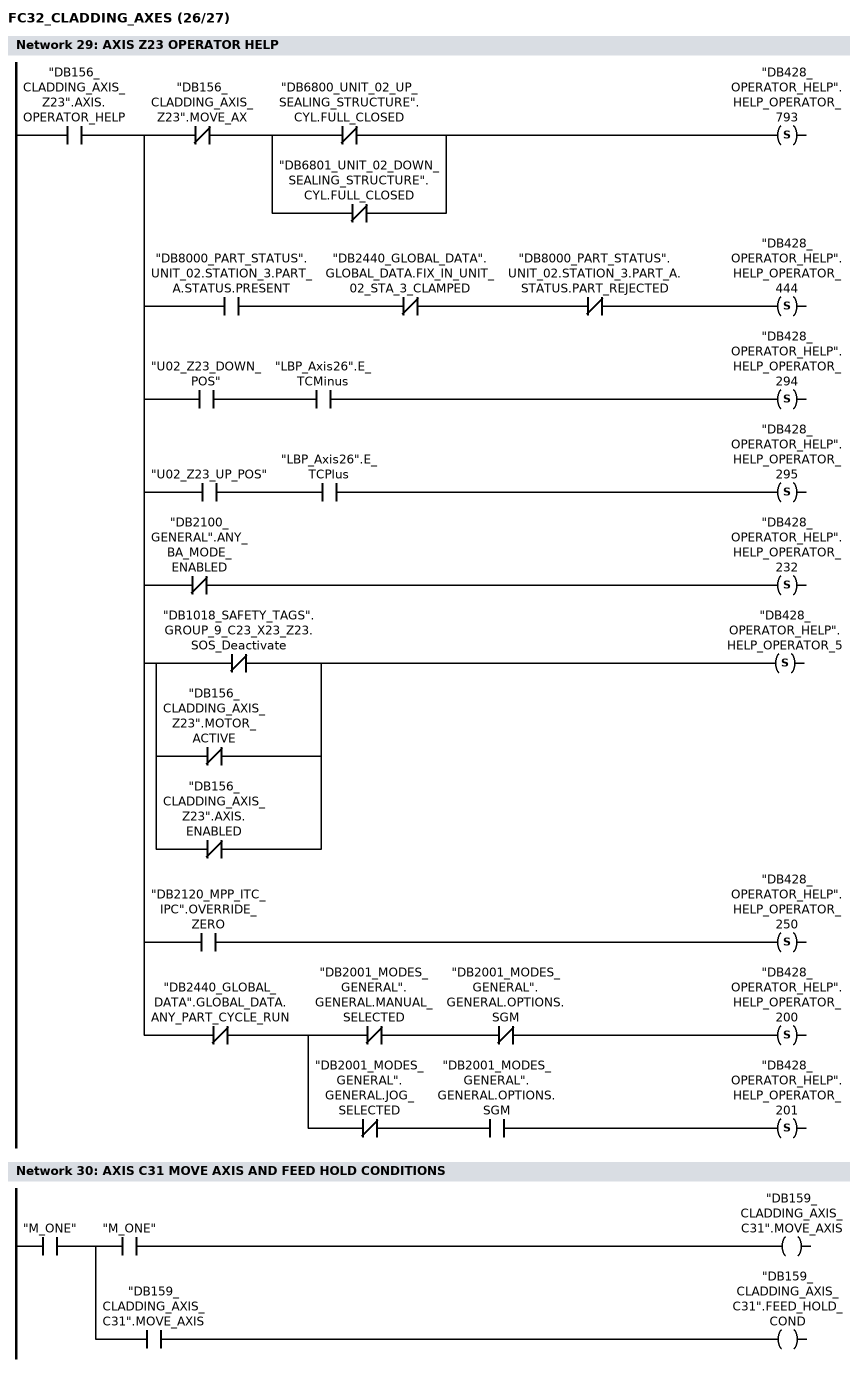
   RUNG wire#powerrail
      Contact( "DB156_CLADDING_AXIS_Z23".AXIS.OPERATOR_HELP )
      wire#w1
      I_Contact( "DB156_CLADDING_AXIS_Z23".MOVE_AX )
      wire#w2
      I_Contact( "DB6800_UNIT_02_UP_SEALING_STRUCTURE".CYL.FULL_CLOSED )
      wire#w3
      S_Coil( "DB428_OPERATOR_HELP".HELP_OPERATOR_793 )
   END_RUNG
   RUNG wire#w2
      I_Contact( "DB6801_UNIT_02_DOWN_SEALING_STRUCTURE".CYL.FULL_CLOSED )
   END_RUNG wire#w3
   RUNG wire#w1
      Contact( "DB8000_PART_STATUS".UNIT_02.STATION_3.PART_A.STATUS.PRESENT )
      I_Contact( "DB2440_GLOBAL_DATA".GLOBAL_DATA.FIX_IN_UNIT_02_STA_3_CLAMPED )
      I_Contact( "DB8000_PART_STATUS".UNIT_02.STATION_3.PART_A.STATUS.PART_REJECTED )
      S_Coil( "DB428_OPERATOR_HELP".HELP_OPERATOR_444 )
   END_RUNG
   RUNG wire#w1
      Contact( "U02_Z23_DOWN_POS" )
      Contact( "LBP_Axis26".E_TCMinus )
      S_Coil( "DB428_OPERATOR_HELP".HELP_OPERATOR_294 )
   END_RUNG
   RUNG wire#w1
      Contact( "U02_Z23_UP_POS" )
      Contact( "LBP_Axis26".E_TCPlus )
      S_Coil( "DB428_OPERATOR_HELP".HELP_OPERATOR_295 )
   END_RUNG
   RUNG wire#w1
      I_Contact( "DB2100_GENERAL".ANY_BA_MODE_ENABLED )
      S_Coil( "DB428_OPERATOR_HELP".HELP_OPERATOR_232 )
   END_RUNG
   RUNG wire#w1
      I_Contact( "DB1018_SAFETY_TAGS".GROUP_9_C23_X23_Z23.SOS_Deactivate )
      wire#w4
      S_Coil( "DB428_OPERATOR_HELP".HELP_OPERATOR_5 )
   END_RUNG
   RUNG wire#w1
      I_Contact( "DB156_CLADDING_AXIS_Z23".MOTOR_ACTIVE )
   END_RUNG wire#w4
   RUNG wire#w1
      I_Contact( "DB156_CLADDING_AXIS_Z23".AXIS.ENABLED )
   END_RUNG wire#w4
   RUNG wire#w1
      Contact( "DB2120_MPP_ITC_IPC".OVERRIDE_ZERO )
      S_Coil( "DB428_OPERATOR_HELP".HELP_OPERATOR_250 )
   END_RUNG
   RUNG wire#w1
      I_Contact( "DB2440_GLOBAL_DATA".GLOBAL_DATA.ANY_PART_CYCLE_RUN )
      wire#w5
      I_Contact( "DB2001_MODES_GENERAL".GENERAL.MANUAL_SELECTED )
      I_Contact( "DB2001_MODES_GENERAL".GENERAL.OPTIONS.SGM )
      S_Coil( "DB428_OPERATOR_HELP".HELP_OPERATOR_200 )
   END_RUNG
   RUNG wire#w5
      I_Contact( "DB2001_MODES_GENERAL".GENERAL.JOG_SELECTED )
      Contact( "DB2001_MODES_GENERAL".GENERAL.OPTIONS.SGM )
      S_Coil( "DB428_OPERATOR_HELP".HELP_OPERATOR_201 )
   END_RUNG
   // the same network as SCL:
   IF "DB156_CLADDING_AXIS_Z23".AXIS.OPERATOR_HELP AND NOT "DB156_CLADDING_AXIS_Z23".MOVE_AX AND (NOT "DB6800_UNIT_02_UP_SEALING_STRUCTURE".CYL.FULL_CLOSED OR NOT "DB6801_UNIT_02_DOWN_SEALING_STRUCTURE".CYL.FULL_CLOSED) THEN
       "DB428_OPERATOR_HELP".HELP_OPERATOR_793 := TRUE;
   END_IF;
   IF "DB156_CLADDING_AXIS_Z23".AXIS.OPERATOR_HELP AND "DB8000_PART_STATUS".UNIT_02.STATION_3.PART_A.STATUS.PRESENT AND NOT "DB2440_GLOBAL_DATA".GLOBAL_DATA.FIX_IN_UNIT_02_STA_3_CLAMPED AND NOT "DB8000_PART_STATUS".UNIT_02.STATION_3.PART_A.STATUS.PART_REJECTED THEN
       "DB428_OPERATOR_HELP".HELP_OPERATOR_444 := TRUE;
   END_IF;
   IF "DB156_CLADDING_AXIS_Z23".AXIS.OPERATOR_HELP AND "U02_Z23_DOWN_POS" AND "LBP_Axis26".E_TCMinus THEN
       "DB428_OPERATOR_HELP".HELP_OPERATOR_294 := TRUE;
   END_IF;
   IF "DB156_CLADDING_AXIS_Z23".AXIS.OPERATOR_HELP AND "U02_Z23_UP_POS" AND "LBP_Axis26".E_TCPlus THEN
       "DB428_OPERATOR_HELP".HELP_OPERATOR_295 := TRUE;
   END_IF;
   IF "DB156_CLADDING_AXIS_Z23".AXIS.OPERATOR_HELP AND NOT "DB2100_GENERAL".ANY_BA_MODE_ENABLED THEN
       "DB428_OPERATOR_HELP".HELP_OPERATOR_232 := TRUE;
   END_IF;
   IF "DB156_CLADDING_AXIS_Z23".AXIS.OPERATOR_HELP AND (NOT "DB1018_SAFETY_TAGS".GROUP_9_C23_X23_Z23.SOS_Deactivate OR NOT "DB156_CLADDING_AXIS_Z23".MOTOR_ACTIVE OR NOT "DB156_CLADDING_AXIS_Z23".AXIS.ENABLED) THEN
       "DB428_OPERATOR_HELP".HELP_OPERATOR_5 := TRUE;
   END_IF;
   IF "DB156_CLADDING_AXIS_Z23".AXIS.OPERATOR_HELP AND "DB2120_MPP_ITC_IPC".OVERRIDE_ZERO THEN
       "DB428_OPERATOR_HELP".HELP_OPERATOR_250 := TRUE;
   END_IF;
   #_w1 := "DB156_CLADDING_AXIS_Z23".AXIS.OPERATOR_HELP AND NOT "DB2440_GLOBAL_DATA".GLOBAL_DATA.ANY_PART_CYCLE_RUN;
   IF #_w1 AND NOT "DB2001_MODES_GENERAL".GENERAL.MANUAL_SELECTED AND NOT "DB2001_MODES_GENERAL".GENERAL.OPTIONS.SGM THEN
       "DB428_OPERATOR_HELP".HELP_OPERATOR_200 := TRUE;
   END_IF;
   IF #_w1 AND NOT "DB2001_MODES_GENERAL".GENERAL.JOG_SELECTED AND "DB2001_MODES_GENERAL".GENERAL.OPTIONS.SGM THEN
       "DB428_OPERATOR_HELP".HELP_OPERATOR_201 := TRUE;
   END_IF;
END_REGION

REGION Network 30: AXIS C31 MOVE AXIS AND FEED HOLD CONDITIONS
   RUNG wire#powerrail
      Contact( "M_ONE" )
      wire#w1
      Contact( "M_ONE" )
      Coil( "DB159_CLADDING_AXIS_C31".MOVE_AXIS )
   END_RUNG
   RUNG wire#w1
      Contact( "DB159_CLADDING_AXIS_C31".MOVE_AXIS )
      Coil( "DB159_CLADDING_AXIS_C31".FEED_HOLD_COND )
   END_RUNG
   // the same network as SCL:
   "DB159_CLADDING_AXIS_C31".MOVE_AXIS := "M_ONE" AND "M_ONE";
   "DB159_CLADDING_AXIS_C31".FEED_HOLD_COND := "M_ONE" AND "DB159_CLADDING_AXIS_C31".MOVE_AXIS;
END_REGION

REGION Network 31: CALL FB32 AXIS C31
   // 2#0000_0001 OPTIONS 0 BIT 0 MEASURING SYSTEM 2 OPTION
   // 2#0000_0010 OPTIONS 0 BIT 1 ENABLE FC18 OPTION
   // 2#0000_0100 OPTIONS 0 BIT 2 FC18 EXTERNAL POSITION OPTION
   // 2#0000_1000 OPTIONS 0 BIT 3 AXIS B ENABLE FAULTS OPTION
   // 2#0001_0000 OPTIONS 0 BIT 4 SPARE OPTION
   // 2#0010_0000 OPTIONS 0 BIT 5 SPARE OPTION
   // 2#0100_0000 OPTIONS 0 BIT 6 SPARE OPTION
   // 2#1000_0000 OPTIONS 0 BIT 7 SPARE OPTION
   // 
   // 2#0000_0001 OPTIONS 1 BIT 0 AXIS ROLLER OPTION
   // 2#0000_0010 OPTIONS 1 BIT 1 MASTER AXIS OPTION
   // 2#0000_0100 OPTIONS 1 BIT 2 SLAVE AXIS OPTION
   // 2#0000_1000 OPTIONS 1 BIT 3 MASTER-SLAVE AXES INDEPENDENT MOVEMENT WITH HT10 OPTION
   // 2#0001_0000 OPTIONS 1 BIT 4 GANTRY MODE MASTER AXIS OPTION
   // 2#0010_0000 OPTIONS 1 BIT 5 SPARE OPTION
   // 2#0100_0000 OPTIONS 1 BIT 6 SPARE OPTION
   // 2#1000_0000 OPTIONS 1 BIT 7 SPARE OPTION
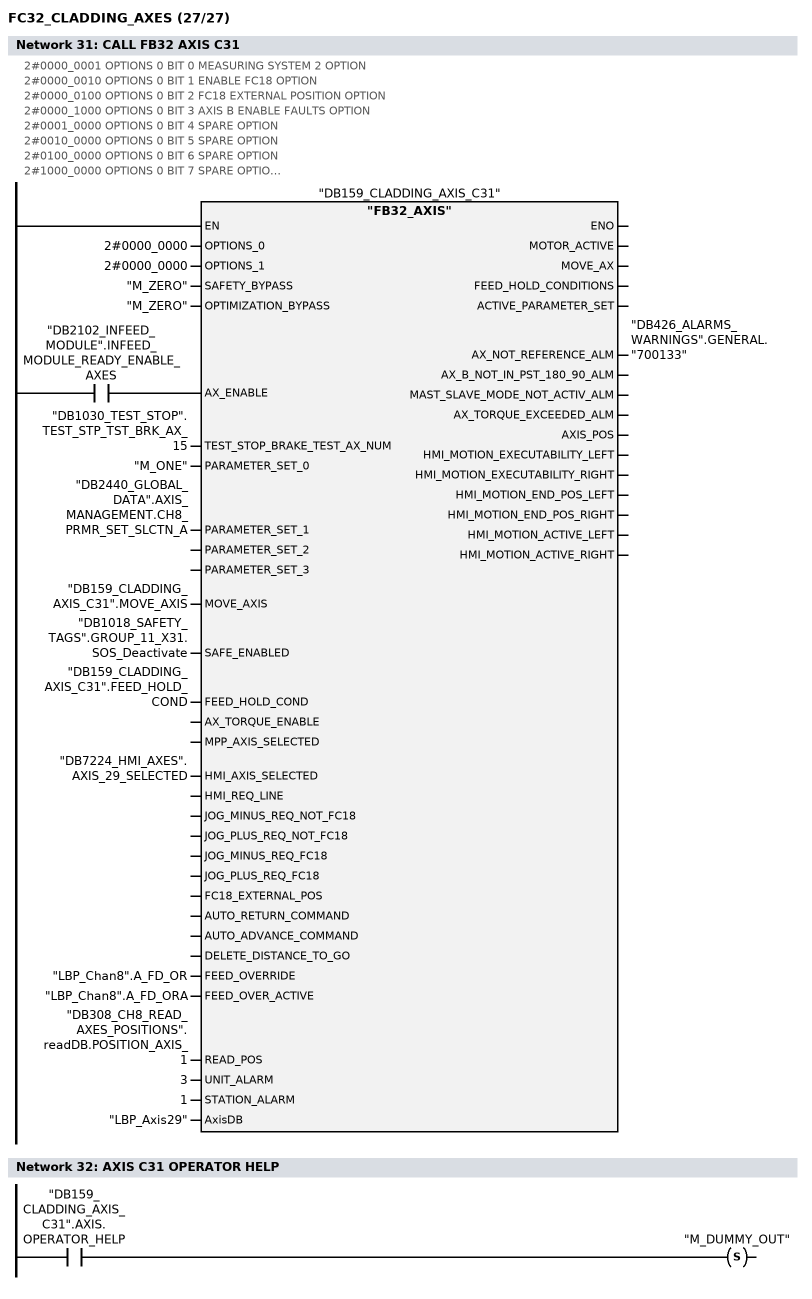
   RUNG wire#powerrail
      "DB159_CLADDING_AXIS_C31"(AX_ENABLE := wire#w1, OPTIONS_0 := 2#0000_0000, OPTIONS_1 := 2#0000_0000, SAFETY_BYPASS := "M_ZERO", OPTIMIZATION_BYPASS := "M_ZERO", TEST_STOP_BRAKE_TEST_AX_NUM := "DB1030_TEST_STOP".TEST_STP_TST_BRK_AX_15, PARAMETER_SET_0 := "M_ONE", PARAMETER_SET_1 := "DB2440_GLOBAL_DATA".AXIS_MANAGEMENT.CH8_PRMR_SET_SLCTN_A, PARAMETER_SET_2 :=, PARAMETER_SET_3 :=, MOVE_AXIS := "DB159_CLADDING_AXIS_C31".MOVE_AXIS, SAFE_ENABLED := "DB1018_SAFETY_TAGS".GROUP_11_X31.SOS_Deactivate, FEED_HOLD_COND := "DB159_CLADDING_AXIS_C31".FEED_HOLD_COND, AX_TORQUE_ENABLE :=, MPP_AXIS_SELECTED :=, HMI_AXIS_SELECTED := "DB7224_HMI_AXES".AXIS_29_SELECTED, HMI_REQ_LINE :=, JOG_MINUS_REQ_NOT_FC18 :=, JOG_PLUS_REQ_NOT_FC18 :=, JOG_MINUS_REQ_FC18 :=, JOG_PLUS_REQ_FC18 :=, FC18_EXTERNAL_POS :=, AUTO_RETURN_COMMAND :=, AUTO_ADVANCE_COMMAND :=, DELETE_DISTANCE_TO_GO :=, FEED_OVERRIDE := "LBP_Chan8".A_FD_OR, FEED_OVER_ACTIVE := "LBP_Chan8".A_FD_ORA, READ_POS := "DB308_CH8_READ_AXES_POSITIONS".readDB.POSITION_AXIS_1, UNIT_ALARM := 3, STATION_ALARM := 1, AxisDB := "LBP_Axis29", MOTOR_ACTIVE =>, MOVE_AX =>, FEED_HOLD_CONDITIONS =>, ACTIVE_PARAMETER_SET =>, AX_NOT_REFERENCE_ALM => "DB426_ALARMS_WARNINGS".GENERAL."700133", AX_B_NOT_IN_PST_180_90_ALM =>, MAST_SLAVE_MODE_NOT_ACTIV_ALM =>, AX_TORQUE_EXCEEDED_ALM =>, AXIS_POS =>, HMI_MOTION_EXECUTABILITY_LEFT =>, HMI_MOTION_EXECUTABILITY_RIGHT =>, HMI_MOTION_END_POS_LEFT =>, HMI_MOTION_END_POS_RIGHT =>, HMI_MOTION_ACTIVE_LEFT =>, HMI_MOTION_ACTIVE_RIGHT =>)
   END_RUNG
   RUNG wire#powerrail
      Contact( "DB2102_INFEED_MODULE".INFEED_MODULE_READY_ENABLE_AXES )
   END_RUNG wire#w1
   // the same network as SCL:
   "DB159_CLADDING_AXIS_C31"(OPTIONS_0 := 2#0000_0000,   // "FB32_AXIS"
                           OPTIONS_1 := 2#0000_0000,
                           SAFETY_BYPASS := "M_ZERO",
                           OPTIMIZATION_BYPASS := "M_ZERO",
                           AX_ENABLE := "DB2102_INFEED_MODULE".INFEED_MODULE_READY_ENABLE_AXES,
                           TEST_STOP_BRAKE_TEST_AX_NUM := "DB1030_TEST_STOP".TEST_STP_TST_BRK_AX_15,
                           PARAMETER_SET_0 := "M_ONE",
                           PARAMETER_SET_1 := "DB2440_GLOBAL_DATA".AXIS_MANAGEMENT.CH8_PRMR_SET_SLCTN_A,
                           MOVE_AXIS := "DB159_CLADDING_AXIS_C31".MOVE_AXIS,
                           SAFE_ENABLED := "DB1018_SAFETY_TAGS".GROUP_11_X31.SOS_Deactivate,
                           FEED_HOLD_COND := "DB159_CLADDING_AXIS_C31".FEED_HOLD_COND,
                           HMI_AXIS_SELECTED := "DB7224_HMI_AXES".AXIS_29_SELECTED,
                           FEED_OVERRIDE := "LBP_Chan8".A_FD_OR,
                           FEED_OVER_ACTIVE := "LBP_Chan8".A_FD_ORA,
                           READ_POS := "DB308_CH8_READ_AXES_POSITIONS".readDB.POSITION_AXIS_1,
                           UNIT_ALARM := 3,
                           STATION_ALARM := 1,
                           AxisDB := "LBP_Axis29",
                           AX_NOT_REFERENCE_ALM => "DB426_ALARMS_WARNINGS".GENERAL."700133");
END_REGION

REGION Network 32: AXIS C31 OPERATOR HELP
   RUNG wire#powerrail
      Contact( "DB159_CLADDING_AXIS_C31".AXIS.OPERATOR_HELP )
      S_Coil( "M_DUMMY_OUT" )
   END_RUNG
   // the same network as SCL:
   IF "DB159_CLADDING_AXIS_C31".AXIS.OPERATOR_HELP THEN "M_DUMMY_OUT" := TRUE; END_IF;
END_REGION
END_FUNCTION
